// Mitsubishi GX Works2 project: mcr_cj   PLC: Q02/Q02H

PROGRAM MCRintro
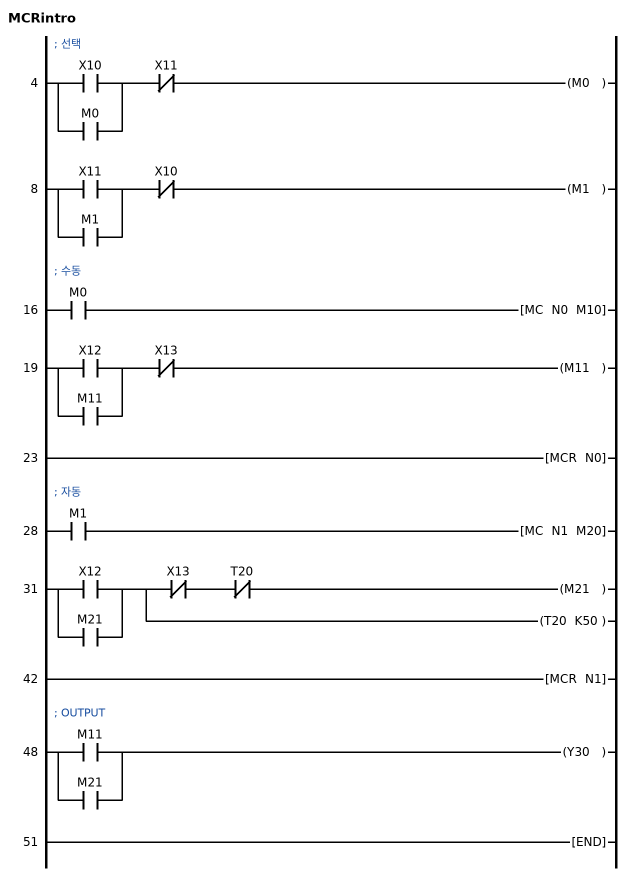
; 선택
4     LD      X10
      OR      M0
      ANI     X11
      OUT     M0
8     LD      X11
      OR      M1
      ANI     X10
      OUT     M1
; 수동
16    LD      M0
      MC      N0 M10
19    LD      X12
      OR      M11
      ANI     X13
      OUT     M11
23    MCR     N0
; 자동
28    LD      M1
      MC      N1 M20
31    LD      X12
      OR      M21
      MPS
      ANI     X13
      ANI     T20
      OUT     M21
      MPP
      OUT     T20 K50
42    MCR     N1
; OUTPUT
48    LD      M11
      OR      M21
      OUT     Y30
51    END
END_PROGRAM

PROGRAM MAIN1
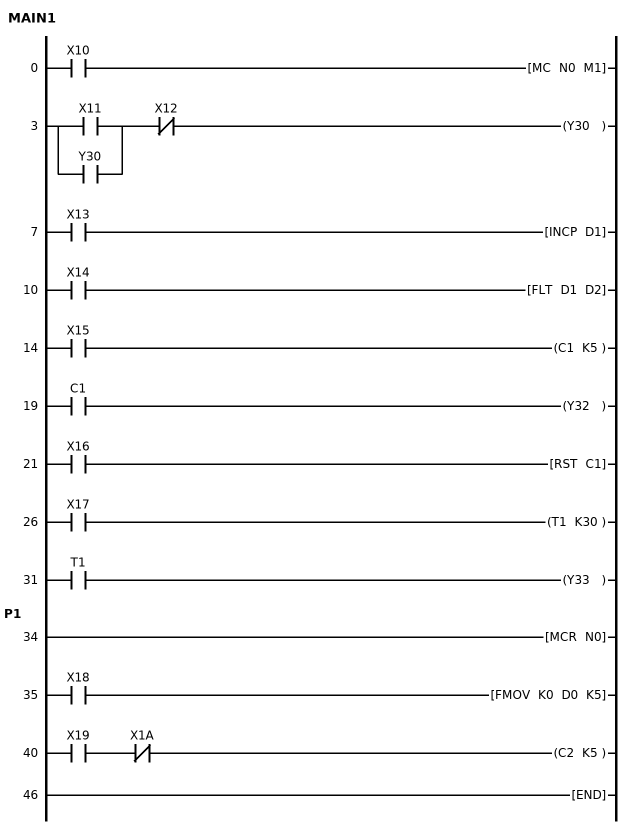
0     LD      X10
      MC      N0 M1
3     LD      X11
      OR      Y30
      ANI     X12
      OUT     Y30
7     LD      X13
      INCP    D1
10    LD      X14
      FLT     D1 D2
14    LD      X15
      OUT     C1 K5
19    LD      C1
      OUT     Y32
21    LD      X16
      RST     C1
26    LD      X17
      OUT     T1 K30
31    LD      T1
      OUT     Y33
      P1
34    MCR     N0
35    LD      X18
      FMOV    K0 D0 K5
40    LD      X19
      ANI     X1A
      OUT     C2 K5
46    END
END_PROGRAM
